INTERFACE ITF_UpdaterRegistry

METHOD Reset : BOOL
VAR_INPUT
END_VAR
END_METHOD

METHOD ResolveUpdater : ITF_Updater
VAR_INPUT
	TypeID	: BYTE;
	Version	: BYTE;
END_VAR
END_METHOD

METHOD TryRegister : HRESULT
VAR_INPUT
	Updater	: ITF_Updater;
END_VAR
END_METHOD

END_INTERFACE

(* stored: Version 1.1.0.1
   Itf ITF_UpdaterRegistry: Id {f37cc204-c2fb-42fe-8f63-27e01e348367}
   Method Reset: Id {3d47ab56-9699-4dea-832d-1e85d8cbf5b0}
   Method ResolveUpdater: Id {c18c0931-7b96-4f34-ade5-921aecccfcd3}
   Method TryRegister: Id {1104802e-94bb-4466-a7d4-8338d9ec9f5f} *)
